// TIA Portal V18 export
DATA_BLOCK "test"   // DB10
{ S7_Optimized_Access := 'TRUE' }
// stored: MemoryReserve 100
   VAR
      statRecord : Array[0..1] of Byte;
      Start : Bool;
      "0R_1W" : Bool;
      Index : Int := 16#41;
      SubIndex : Int;
      LEN : Int := 2;
      diag : "LIOLink_typeDiagnostics";
   END_VAR
BEGIN
END_DATA_BLOCK
